// TIA Portal project "RemoteConection" (V20)

(* hardware
DEVICE "S7-1500/ET200MP station_1"  S7-1500 station
   slot 0: "Rail_0"  Rack  6ES7 590-1***0-0AA0
   slot 1: "PLC_1"  CPU 1518-4 PN/DP  6ES7 518-4AP00-0AB0  V3.1
      slot 3: "CPU display_1"  6ES7591-1BA00-0AA0
      slot 32768: "PROFINET interface_1"  X1
         slot 32769: "Port_1"  X1 P1
         slot 32770: "Port_2"  X1 P2
      slot 33024: "PROFINET interface_2"  X2
         slot 33025: "Port_1"  X2 P1
      slot 33280: "PROFINET interface GBIT_3"  X3
         slot 33281: "Port_1"  X3 P1
      slot 33536: "DP interface_1"  X4
      slot 34817: "Virtual CP interface port_1"  Virtual CP interface port  Virtual CP interface port
   slot 2: "DI 16x24VDC HF_1"  DI 16x24VDC HF  6ES7 521-1BH00-0AB0  V2.2
   slot 3: "DQ 16x24VDC/0.5A HF_1"  DQ 16x24VDC/0.5A HF  6ES7 522-1BH01-0AB0  V1.1
*)

// ===== PLC "PLC_1"  CPU 1518-4 PN/DP =====

VAR_GLOBAL   // PLC tag table "Default tag table"
   "Clock_Byte" AT %MB10 : Byte;
   "Clock_10Hz" AT %M10.0 : Bool;
   "Clock_5Hz" AT %M10.1 : Bool;
   "Clock_2.5Hz" AT %M10.2 : Bool;
   "Clock_2Hz" AT %M10.3 : Bool;
   "Clock_1.25Hz" AT %M10.4 : Bool;
   "Clock_1Hz" AT %M10.5 : Bool;
   "Clock_0.625Hz" AT %M10.6 : Bool;
   "Clock_0.5Hz" AT %M10.7 : Bool;
END_VAR

DATA_BLOCK "RemoteConnection"   // DB1
{ S7_Optimized_Access := 'TRUE' }
VERSION : 0.1
   VAR
      Out : Int;
      Write : Int;
   END_VAR
BEGIN
END_DATA_BLOCK

DATA_BLOCK "Block_1_DB"   // DB2
{ S7_Optimized_Access := 'TRUE' }
VERSION : 0.1
// stored: InstanceOfName Block_1
"Block_1"
BEGIN
END_DATA_BLOCK

DATA_BLOCK "Semaforo_RM_DB"   // DB3
{ S7_Optimized_Access := 'TRUE' }
VERSION : 0.1
// stored: InstanceOfName Semaforo_RM
"Semaforo_RM"
BEGIN
END_DATA_BLOCK

DATA_BLOCK "Semaforo_RM2"   // DB4
{ S7_Optimized_Access := 'TRUE' }
VERSION : 0.1
   VAR
      f_prueba : Bool;
      start : Bool;
      stop : Bool;
      f_rojo : Bool;
      f_amarillo : Bool;
      f_verde : Bool;
      current_time : Time;
   END_VAR
BEGIN
END_DATA_BLOCK

FUNCTION_BLOCK "Block_1"   // FB1, LAD
{ S7_Optimized_Access := 'TRUE' }
VERSION : 0.1
   VAR_OUTPUT
      Out : USInt;
   END_VAR
   VAR
      Tiempo : UDInt;
      "Mod" : UDInt;
      Div : UDInt;
   END_VAR
BEGIN

REGION Network 1
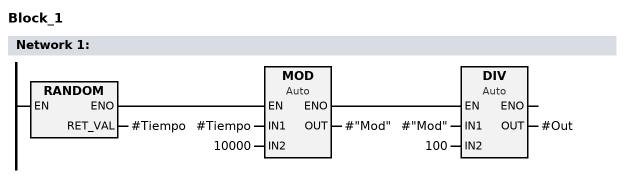
   // no SCL statement known for Random: written as a call
   // ENO of a box is taken as its EN; it also drops when the box reports an error
   #Tiempo := Random();
   #"Mod" := #Tiempo MOD 10000;
   #Out := #"Mod" / 100;
END_REGION
END_FUNCTION_BLOCK

FUNCTION_BLOCK "Semaforo_RM"   // FB2, LAD
{ S7_Optimized_Access := 'TRUE' }
VERSION : 0.1
   VAR_INPUT
      inicio : Bool;
      stop : Bool;
   END_VAR
   VAR_OUTPUT
      f_rojo : Bool;
      f_amarillo : Bool;
      f_verde : Bool;
      prueba : Bool;
      tiempo_restante : Time;
   END_VAR
   VAR
      t_rojo : Bool;
      t_amarillo : Bool;
      t_verde : Bool;
      paso_ : Bool;
      paso_2 : Bool;
      c_rojo : IEC_TIMER;
      c_amarillo : IEC_TIMER;
      c_verde : IEC_TIMER;
      time_rojo : Time := T#7s;
      time_amarillo : Time := T#5s;
      time_verde : Time := T#15s;
      et_rojo : Time;
      et_amarillo : Time;
      et_verde : Time;
      enc_t_rojo : Bool;
      enc_t_amarillo : Bool;
      enc_t_verde : Bool;
      enc_t_intermitente : Bool;
      enc_start : Bool;
      enc_aux : Bool;
   END_VAR
   VAR_TEMP   // added for the SCL form of the ladder/FBD networks
      _w1 : Bool;
      _w2 : Bool;
   END_VAR
BEGIN

REGION Network 1
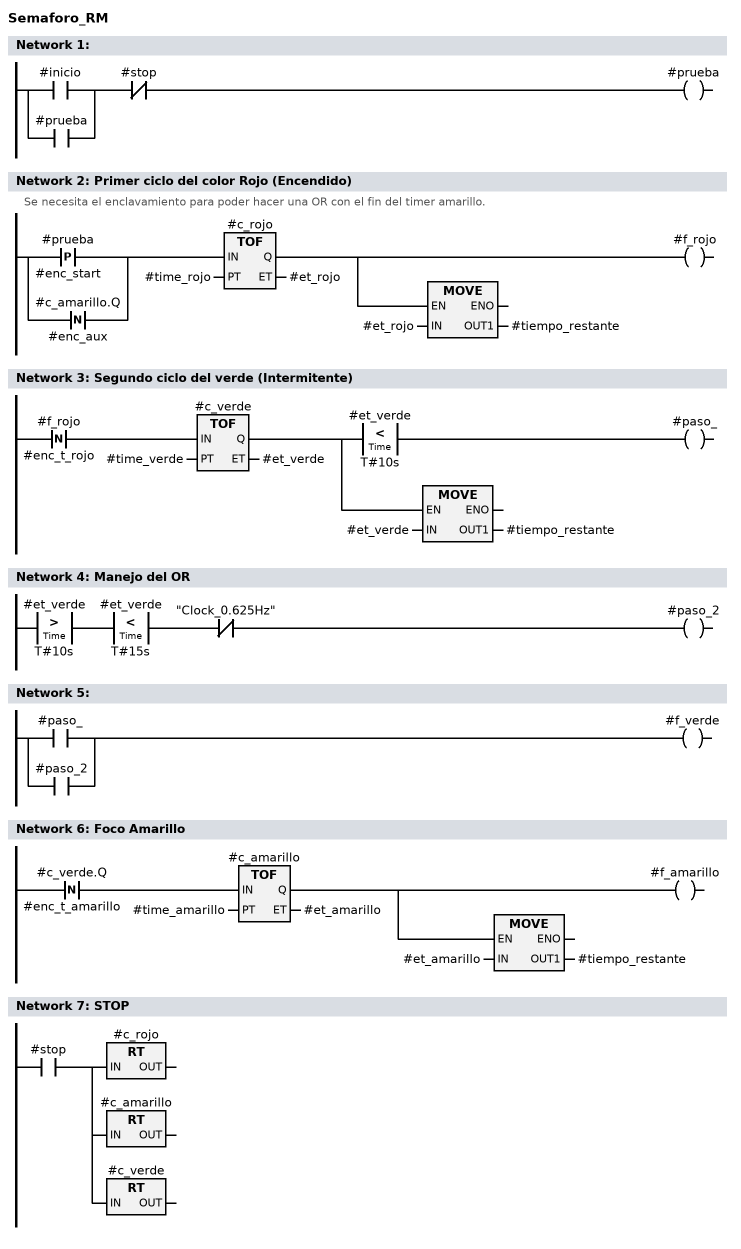
   RUNG wire#powerrail
      Contact( #inicio )
      wire#w1
      I_Contact( #stop )
      Coil( #prueba )
   END_RUNG
   RUNG wire#powerrail
      Contact( #prueba )
   END_RUNG wire#w1
   // the same network as SCL:
   #prueba := (#inicio OR #prueba) AND NOT #stop;
END_REGION

REGION Network 2: Primer ciclo del color Rojo (Encendido)
   // Se necesita el enclavamiento para poder hacer una OR con el fin del timer amarillo.
   #_w1 := #prueba AND NOT #enc_start;   // rising edge of #prueba
   #enc_start := #prueba;
   #_w2 := NOT #c_amarillo.Q AND #enc_aux;   // falling edge of #c_amarillo.Q
   #enc_aux := #c_amarillo.Q;
   #c_rojo.TOF(IN := #_w1 OR #_w2, PT := #time_rojo, ET => #et_rojo);
   #f_rojo := #c_rojo.Q;
   IF #c_rojo.Q THEN #tiempo_restante := #et_rojo; END_IF;
END_REGION

REGION Network 3: Segundo ciclo del verde (Intermitente)
   #_w1 := NOT #f_rojo AND #enc_t_rojo;   // falling edge of #f_rojo
   #enc_t_rojo := #f_rojo;
   #c_verde.TOF(IN := #_w1, PT := #time_verde, ET => #et_verde);
   #paso_ := #c_verde.Q AND (#et_verde < T#10s);
   IF #c_verde.Q THEN #tiempo_restante := #et_verde; END_IF;
END_REGION

REGION Network 4: Manejo del OR
   RUNG wire#powerrail
      { S7_Templates := "SrcType := Time" } GT_Contact(in1 := #et_verde, in2 := T#10s)
      { S7_Templates := "SrcType := Time" } LT_Contact(in1 := #et_verde, in2 := T#15s)
      I_Contact( "Clock_0.625Hz" )
      Coil( #paso_2 )
   END_RUNG
   // the same network as SCL:
   #paso_2 := (#et_verde > T#10s) AND (#et_verde < T#15s) AND NOT "Clock_0.625Hz";
END_REGION

REGION Network 5
   RUNG wire#powerrail
      Contact( #paso_ )
      wire#w1
      Coil( #f_verde )
   END_RUNG
   RUNG wire#powerrail
      Contact( #paso_2 )
   END_RUNG wire#w1
   // the same network as SCL:
   #f_verde := #paso_ OR #paso_2;
END_REGION

REGION Network 6: Foco Amarillo
   #_w1 := NOT #c_verde.Q AND #enc_t_amarillo;   // falling edge of #c_verde.Q
   #enc_t_amarillo := #c_verde.Q;
   #c_amarillo.TOF(IN := #_w1, PT := #time_amarillo, ET => #et_amarillo);
   #f_amarillo := #c_amarillo.Q;
   IF #c_amarillo.Q THEN #tiempo_restante := #et_amarillo; END_IF;
END_REGION

REGION Network 7: STOP
   RUNG wire#powerrail
      Contact( #stop )
      wire#w1
      RT_Coil( #c_rojo )
   END_RUNG
   RUNG wire#w1
      RT_Coil( #c_amarillo )
   END_RUNG
   RUNG wire#w1
      RT_Coil( #c_verde )
   END_RUNG
   // the same network as SCL:
   IF #stop THEN
       RESET_TIMER(#c_rojo);
       RESET_TIMER(#c_amarillo);
       RESET_TIMER(#c_verde);
   END_IF;
END_REGION
END_FUNCTION_BLOCK

ORGANIZATION_BLOCK "Main"   // OB1, LAD, ProgramCycle
TITLE = "Main Program Sweep (Cycle)"
{ S7_Optimized_Access := 'TRUE' }
VERSION : 0.1
   VAR_INPUT
      Initial_Call : Bool;   // Initial call of this OB
      Remanence : Bool;   // =True, if remanent data are available
   END_VAR
BEGIN

REGION Network 1
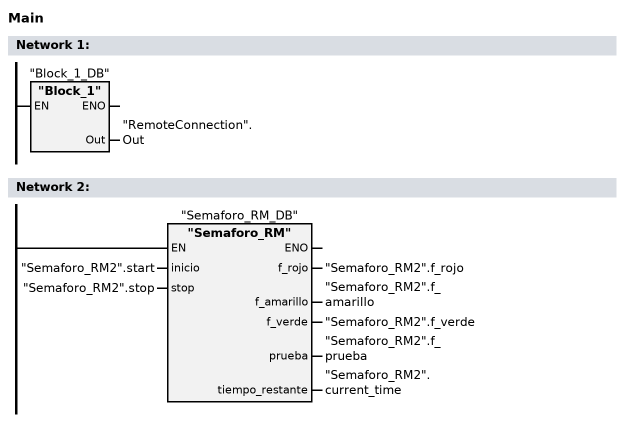
   RUNG wire#powerrail
      "Block_1_DB"(Out => "RemoteConnection".Out)
   END_RUNG
   // the same network as SCL:
   "Block_1_DB"(Out => "RemoteConnection".Out);   // "Block_1"
END_REGION

REGION Network 2
   RUNG wire#powerrail
      "Semaforo_RM_DB"(inicio := "Semaforo_RM2".start, stop := "Semaforo_RM2".stop, f_rojo => "Semaforo_RM2".f_rojo, f_amarillo => "Semaforo_RM2".f_amarillo, f_verde => "Semaforo_RM2".f_verde, prueba => "Semaforo_RM2".f_prueba, tiempo_restante => "Semaforo_RM2".current_time)
   END_RUNG
   // the same network as SCL:
   "Semaforo_RM_DB"(inicio := "Semaforo_RM2".start,   // "Semaforo_RM"
                    stop := "Semaforo_RM2".stop,
                    f_rojo => "Semaforo_RM2".f_rojo,
                    f_amarillo => "Semaforo_RM2".f_amarillo,
                    f_verde => "Semaforo_RM2".f_verde,
                    prueba => "Semaforo_RM2".f_prueba,
                    tiempo_restante => "Semaforo_RM2".current_time);
END_REGION
END_ORGANIZATION_BLOCK